Universal Robots PolyScope program: andrea6.urp

Program andrea6 (installation=Kong_install directory=/home/ur/ursim-current/programs/andrea6 createdIn=3.15.4.106291 lastSavedIn=3.15.4.106291 robotSerialNumber=2018359999)
Calibrated DH parameters: a=[0.000104, -0.381245, -0.385946, 0.00002, 0.000083, 0]; d=[0.089177, 59.99214, -36.297918, -23.584132, 0.094784, 0.082552]; alpha=[1.570197, -0.003145, 0.002952, 1.570494, -1.570091, 0]; deltaTheta=[-0.00001, -0.459739, 0.638868, -0.17972, -0.000006, -0.000462]
InitVariablesNode variables(variable(name=XY, expression=[0,0]), variable(name=nCycle, expression=0), variable(name=pallStocks, expression=[16,16,16,40,16,16,16,40,16,16,16,40,16,40,0,0]), variable(name=pick, expression=[0,0]))
Robot Program (runOnlyOnce=false)
  Script file /home/ur/ursim-current/programs/relPose.script
    | def relPose(FeaturePose,vect):
    | 
    |     # FeaturePose is the pose for the feature
    |     # vect = p[0.1, 0, 0, 0, 0, 0] makes us move 10cm in the X direction of the feature
    |     # credits: https://forum.universal-robots.com/t/move-tcp-relative-to-feature/15492
    | 
    |    PoseRelativeToFeature = pose_trans(pose_inv(FeaturePose), get_actual_tcp_pose())
    |    MoveTCPRelativeToFeature = pose_add(PoseRelativeToFeature, vect)
    |    return pose_trans(FeaturePose, MoveTCPRelativeToFeature)
    | 
    | end
  Script file /home/ur/ursim-current/programs/andrea5/calcItemPosition.script
    | def calcItemPosition(pick, item, pallDefs, grid):
    | 
    |     # calcola la posizione assoluta del pezzo scelto da pickPalletItem
    |     # l'origine è considerato il punto 0 del primo slot della griglia
    | 
    |     # nPosX è il numero di colonne
    |     # nPosY è il numero di righe
    |     # distX è la distanza tra colonne
    |     # distY è la distanza tra righe
    |     # [posX1, posY1] è la posizione del primo pezzo rispetto all'origine del pallet
    | 
    |     nPallet = pick[0] + 1 # numero del pallet (gli id partono da 0)
    |     nItem = pick[1] + 1 # numero del pezzo
    | 
    |     nPosXgrid = grid[0] # numero di posizioni della giglia in X
    |     distXgrid = grid[2] # distanza tra gli slot della griglia in X
    |     distYgrid = grid[3] # distanza tra gli slot della griglia in Y
    | 
    |     pallPosX = nPallet%nPosXgrid
    |     if(pallPosX==0): pallPosX = nPosXgrid end
    |     pallPosY = ceil(nPallet/nPosXgrid)
    | 
    |     nPosX = pallDefs[item,0]
    |     nPosY = pallDefs[item,1]
    |     distX = pallDefs[item,2]
    |     distY = pallDefs[item,3]
    |     posX1 = pallDefs[item,4]
    |     posY1 = pallDefs[item,5]
    | 
    |     posX = nItem%nPosX
    |     if(posX==0): posX = nPosX end
    |     posY = ceil(nItem/nPosX)
    | 
    |     # [X,Y] è la posizione del pezzo rispetto all'origine della griglia
    | 
    |     X=distX*(posX - 1) + posX1 + distXgrid*(pallPosX - 1)
    |     Y=distY*(posY - 1) + posY1 + distYgrid*(pallPosY - 1)
    |     xy=[X,Y]
    | 
    |     return xy
    | 
    |  end
  Script file /home/ur/ursim-current/programs/andrea5/pickPalletItem.script
    | def pickPalletItem(type, pallDefs, pallTypes, pallStocks):
    | 
    |   # seleziona un pezzo sulla griglia, noti il tipo di pezzo e lo stato della griglia
    | 
    |   # lo script funziona finché le variabili del robot non vengono resettate. Tuttavia, anche
    |   # in caso di riavvio, è possibile scrivere manualmente le info sulla griglia e lo stock
    |   # all'inizio del programma, così da 'insegnare' al robot dove farlo
    |   # riprendere
    | 
    |   iPallet = 0 # inizializzo l'id del pallet
    | 
    |   while iPallet < length(pallStocks):
    | 
    |     if pallTypes[iPallet] == type and pallStocks[iPallet] > 0 :
    | 
    |       nItems = pallStocks[iPallet] # numero di pezzi nello stock del pallet iesimo
    | 
    |       nPosX = pallDefs[type,0] # numero di posizioni lungo x, come definito per il pallet di tipo "type"
    |       nPosY = pallDefs[type,1] # numero di posizioni lungo y, come definito per il pallet di tipo "type"
    | 
    |       stockMax = nPosX*nPosY
    |       iItem = stockMax - nItems # id del pezzo
    | 
    |       pick = [iPallet,iItem]
    | 
    |       # pick = [id del pallet, id del pezzo]
    | 
    |       return pick
    |  end
    | iPallet = iPallet + 1
    | end
    | end
  Script file /home/ur/ursim-current/programs/andrea_mk2/stockUpdate.script
    | def stockUpdate(pick,stock):
    | 
    |     # simple function that ingests the output of pickItem and returns the
    |     # modified stock array. just so to avoid using global variables and
    |     # multi-dimensional arrays
    | 
    |     i = pick[0]
    |     stock[i] = stock[i] - 1
    |     return stock
    | 
    | 
    | end
  Script file /home/ur/ursim-current/programs/andrea6/ini_grid.script
    | def ini_grid():
    | 
    |     grid = [4,4,90,90]
    |     return grid
    | end
  Script file /home/ur/ursim-current/programs/andrea6/ini_defs.script
    | def ini_defs():
    | 
    |     # definition = [nPosX,nPosY,distX,distY,posX1,posY1]
    | 
    |     # nPosX è il numero di colonne
    |     # nPosY è il numero di righe
    |     # distX è la distanza tra colonne
    |     # distY è la distanza tra righe
    |     # [posX1, posY1] è la posizione del primo pezzo rispetto all'origine del pallet
    | 
    |     defs = [
    |         [0,0,0,0,0,0], # slot vuoto
    |         [4,10,18,8,16.42,19.06], # pallet nfc
    |         [4,4,22,22,11,11] # pallet ghiere
    |     ]
    |     return defs
    | end
  Script file /home/ur/ursim-current/programs/andrea6/ini_types.script
    | def ini_types():
    | 
    |     visualTypes = [
    | 
    |         [2,1,0,0],
    |         [2,2,2,1],
    |         [2,2,2,1],
    |         [2,2,2,1]
    | 
    |     ]
    | 
    | # purtroppo fare questa array vuota di dimensione (righe)x(colonne) per aggirare le limitazioni di UR
    | # bisogna ricordarsi di cambiare questa dichiarazione di types se si cambia dimensione griglia
    | 
    |      types = [0,0,0,0,0,0,0,0,0,0,0,0,0,0,0,0]
    | 
    |     iii = 0
    |     s = size(visualTypes)
    |     i = 0
    |     while i < s[0]:
    | 
    |         ii=0
    |         while ii < s[1]:
    | 
    |             types[iii] = visualTypes[s[0]-1-i,ii]
    |             ii = ii + 1
    |             iii = iii + 1
    |         end
    |     i = i + 1
    |     end
    |     return types
    | end
  Script file /home/ur/ursim-current/programs/andrea6/ini_stocks.script
    | def ini_stocks():
    | 
    | 
    |     visualStocks = [
    | 
    |         [16, 40, 0, 0],
    |         [16, 16, 16, 40],
    |         [16, 16, 16, 40],
    |         [16 ,16, 16, 40]
    | 
    |     ]
    | 
    | # purtroppo fare questa array vuota di dimensione (righe)x(colonne) per aggirare le limitazioni di UR
    | # bisogna ricordarsi di cambiare questa dichiarazione di types se si cambia dimensione griglia
    | 
    |      stocks = [0,0,0,0,0,0,0,0,0,0,0,0,0,0,0,0]
    | 
    |     iii = 0
    |     s = size(visualStocks)
    |     i = 0
    |     while i < s[0]:
    | 
    |         ii=0
    |         while ii < s[1]:
    | 
    |             stocks[iii] = visualStocks[s[0]-1-i,ii]
    |             ii = ii + 1
    |             iii = iii + 1
    |         end
    |     i = i + 1
    |     end
    |     return stocks
    | end
  If nCycle≟0
    pallTypes := ini_types()
    grid := ini_grid()
    pallDefs := ini_defs()
    pallStocks := ini_stocks()
    Popup Message (haltProgram=false inputType=Variable) variable=grid
    nCycle := 1
  MoveJ speed 60 deg/s, acceleration 80 deg/s^2 (useActiveTCP=false) tcp=Ventosa
    SuppressedNode
      Waypoint Waypoint_1: TCP in base x=-127.249 y=569.007 z=-273.97 mm, rx=-2.3039 ry=-0.5206 rz=-0.2288 rad; joints [-88.999, -25.01, 79.358, -9.678, 91.456, 155.199] deg; flange x=-120.447 y=603.545 z=-174.923 mm, rx=-2.3039 ry=-0.5206 rz=-0.2288 rad
    Waypoint azzeramento: TCP in base x=49.535 y=412.362 z=-175.19 mm, rx=-2.2888 ry=-0.6043 rz=-0.263 rad; joints [-113.333, -47.861, 113.708, -18.803, 74.118, 133.37] deg; flange x=49.53 y=447.275 z=-76.04 mm, rx=-2.2888 ry=-0.6043 rz=-0.263 rad
  item := 2
  pick := pickPalletItem(item,pallDefs,pallTypes,pallStocks)
  XY := calcItemPosition(pick, item,pallDefs, grid)
  MoveJ speed 60 deg/s, acceleration 80 deg/s^2 (useActiveTCP=false) tcp=Ventosa
    Popup Message (haltProgram=false inputType=Variable) variable=pick
    SuppressedNode
      Waypoint Waypoint_2: TCP in base x=-58.441 y=489.516 z=-250.08 mm, rx=-2.2888 ry=-0.6043 rz=-0.263 rad; joints [-96.49, -34.009, 98.153, -19.269, 86.152, 145.828] deg; flange x=-58.447 y=524.429 z=-150.93 mm, rx=-2.2888 ry=-0.6043 rz=-0.263 rad
    p_pall := relPose(Piano_Carrello,p[XY[0]/1000,XY[1]/1000,0.0,0.0,0.0,0.0])
    Waypoint Waypoint (Variable): variable=p_pall
    SuppressedNode
      centro_modulo := relPose(Piano_Carrello,p[-0.05,-0.05,0.0,0.0,0.0,0.0])
    SuppressedNode
      Waypoint Waypoint (Variable): variable=centro_modulo
    SuppressedNode
      pezzo1 := relPose(Piano_Carrello,p[-0.0275,-0.0337,0.0,0.0,0.0,0.0])
  MoveL speed 250 mm/s, acceleration 1200 mm/s^2 (useActiveTCP=false) tcp=Ventosa; feature=Base
    SuppressedNode
      Popup Message (haltProgram=false message=o inputType=Text)
    p_pall := relPose(Piano_Carrello,p[0.0,0.0,-0.1,0.0,0.0,0.0])
    Waypoint Waypoint (Variable): variable=p_pall
    p_pall := relPose(Piano_Carrello,p[0.0,0.0,+0.1,0.0,0.0,0.0])
    Waypoint Waypoint (Variable): variable=p_pall
    pallStocks := stockUpdate(pick,pallStocks)
    Popup Message (haltProgram=false inputType=Variable) variable=pallStocks
  SuppressedNode
    MoveJ speed 60 deg/s, acceleration 80 deg/s^2 (useActiveTCP=false) tcp=Ventosa
      Waypoint Punto_percors_1: TCP in base x=360.235 y=592.133 z=-312.029 mm, rx=-2.2888 ry=-0.6043 rz=-0.263 rad; joints [-131.868, -6.111, 42.389, 16.446, 62.296, 118.284] deg; flange x=360.229 y=627.047 z=-212.879 mm, rx=-2.2888 ry=-0.6043 rz=-0.263 rad
      Waypoint Punto_percors_2: TCP in base x=359.846 y=566.873 z=-337.553 mm, rx=-2.2887 ry=-0.6044 rz=-0.2629 rad; joints [-133.35, -6.1, 47.305, 12.155, 61.413, 116.94] deg; flange x=359.84 y=601.783 z=-238.403 mm, rx=-2.2887 ry=-0.6044 rz=-0.2629 rad
      Waypoint Punto_percors_3: TCP in base x=360.405 y=604.095 z=-299.967 mm, rx=-2.2888 ry=-0.6043 rz=-0.2631 rad; joints [-131.197, -5.882, 39.639, 18.687, 62.698, 118.883] deg; flange x=360.394 y=639.008 z=-200.817 mm, rx=-2.2888 ry=-0.6043 rz=-0.2631 rad
      Waypoint Punto_percors_4: TCP in base x=361.884 y=393.627 z=-97.825 mm, rx=-2.3321 ry=-0.5975 rz=-0.2952 rad; joints [-145.924, -43.509, 87.922, 15.491, 57.335, 104.682] deg; flange x=360.373 y=432.103 z=-0.014 mm, rx=-2.3321 ry=-0.5975 rz=-0.2952 rad
  SuppressedNode
    MoveJ speed 60 deg/s, acceleration 80 deg/s^2 (useActiveTCP=false) tcp=Dosatore_Colla
      Waypoint Punto_percors_5: TCP in base x=368.156 y=553.933 z=-129.773 mm, rx=-2.3872 ry=0.0262 rz=-0.0499 rad; joints [-145.925, -43.512, 87.923, 15.491, 57.335, 104.68] deg; flange x=360.385 y=432.094 z=0.008 mm, rx=-2.3321 ry=-0.5975 rz=-0.2952 rad
      Waypoint Punto_percors_6: TCP in base x=346.525 y=429.809 z=-90.901 mm, rx=2.8684 ry=-0.498 rz=0.4963 rad; joints [-130.235, -41.25, 75.1, 55.819, 112.109, 129.678] deg; flange x=294.495 y=472.211 z=74.153 mm, rx=2.8334 ry=0.2554 rz=0.398 rad
      Waypoint Punto_percors_7: TCP in base x=345.7 y=374.489 z=-146.809 mm, rx=2.8685 ry=-0.4978 rz=0.4962 rad; joints [-134.218, -41.871, 86.428, 43.5, 112.047, 125.394] deg; flange x=293.676 y=416.87 z=18.254 mm, rx=2.8335 ry=0.2556 rz=0.3979 rad
      Waypoint Punto_percors_8: TCP in base x=332.241 y=373.424 z=-148.053 mm, rx=2.8953 ry=-0.2434 rz=0.8191 rad; joints [-129.612, -46.561, 97.376, 26.024, 119.722, 116.801] deg; flange x=241.61 y=402.136 z=2.645 mm, rx=2.7481 ry=0.4942 rz=0.7142 rad
      Waypoint Punto_percors_9: TCP in base x=332.91 y=419.209 z=-101.82 mm, rx=2.8952 ry=-0.2434 rz=0.819 rad; joints [-126.246, -46.699, 88.52, 36.923, 120.408, 120.592] deg; flange x=242.285 y=447.932 z=48.879 mm, rx=2.7481 ry=0.4942 rz=0.7141 rad
  SuppressedNode
    MoveJ speed 60 deg/s, acceleration 80 deg/s^2 (useActiveTCP=false) tcp=Ventosa
      Waypoint Punto_percor_10: TCP in base x=247.37 y=347.613 z=17.849 mm, rx=2.7481 ry=0.4942 rz=0.714 rad; joints [-126.247, -46.7, 88.522, 36.924, 120.406, 120.593] deg; flange x=242.286 y=447.918 z=48.877 mm, rx=2.7481 ry=0.4942 rz=0.714 rad
      Waypoint Punto_percor_11: TCP in base x=335.749 y=393.911 z=-97.703 mm, rx=-2.0353 ry=0.1912 rz=-2.0441 rad; joints [-127.274, -47.792, 108.361, -61.985, 138.312, 104.384] deg; flange x=284.356 y=456.498 z=-30.687 mm, rx=-2.0353 ry=0.1912 rz=-2.0441 rad
      Waypoint Punto_percor_12: TCP in base x=338.359 y=373.234 z=-145.029 mm, rx=-1.712 ry=0.6311 rz=-1.7722 rad; joints [-132.228, -47.414, 117.865, -75.373, 134.377, 130.604] deg; flange x=286.4 y=396.013 z=-56.536 mm, rx=-1.712 ry=0.6311 rz=-1.7722 rad
      Waypoint Punto_percor_13: TCP in base x=337.572 y=370.981 z=-149.981 mm, rx=-1.7121 ry=0.6312 rz=-1.7722 rad; joints [-132.354, -46.82, 118.144, -76.237, 134.255, 130.611] deg; flange x=285.617 y=393.768 z=-61.488 mm, rx=-1.7121 ry=0.6312 rz=-1.7722 rad
      Waypoint Punto_percor_12: TCP in base x=338.359 y=373.234 z=-145.029 mm, rx=-1.712 ry=0.6311 rz=-1.7722 rad; joints [-132.228, -47.414, 117.865, -75.373, 134.377, 130.604] deg; flange x=286.4 y=396.013 z=-56.536 mm, rx=-1.712 ry=0.6311 rz=-1.7722 rad
      Waypoint Punto_percor_14: TCP in base x=335.761 y=393.868 z=-97.693 mm, rx=-2.0353 ry=0.1912 rz=-2.0442 rad; joints [-127.277, -47.794, 108.365, -61.99, 138.314, 104.379] deg; flange x=284.372 y=456.463 z=-30.681 mm, rx=-2.0353 ry=0.1912 rz=-2.0442 rad
